(* PLC project Robots Function Blocks, JihuaLab Robots Function Blocks 1.0, author Zebang Zhong *)
(* stored: creationDateTime 2020-02-21T09:44:11, modificationDateTime 2020-04-25T15:42:12 *)

(* This block makes the robot ready. *)
FUNCTION_BLOCK RobotEnable
  VAR_INPUT
    ENABLE : BOOL;  (* TRUE to enable the block *)
    STATE : SINT;  (* Current state of robot *)
  END_VAR
  VAR_OUTPUT
    VALID : BOOL;  (* This is the output shows if robot is enabled *)
  END_VAR

          If ENABLE = TRUE then run
        
END_FUNCTION_BLOCK

(* This block makes the robot ready. *)
FUNCTION_BLOCK MotionGo
  VAR_INPUT
    ENABLE : BOOL;  (* TRUE to enable the block *)
  END_VAR
  VAR_OUTPUT
    VALID : BOOL;  (* This is the output shows if robot is ready *)
  END_VAR

          If ENABLE = TRUE then run
        
END_FUNCTION_BLOCK

(* This block gets the current joints of the robot. *)
FUNCTION_BLOCK GetCurJoint
  VAR_INPUT
    ENABLE : BOOL;  (* TRUE to enable the block *)
  END_VAR
  VAR_OUTPUT
    VALID : BOOL;  (* This is the output shows if result received *)
    ERROR : BOOL;  (* This is the output shows if error occured *)
    ERRORCODE : SINT;  (* This is the output shows the error code *)
    JOINT : STRING;  (* This is the output shows the joints *)
    EXTJOINT : STRING;  (* This is the output shows the extjoints *)
  END_VAR

          If ENABLE = TRUE then run
        
END_FUNCTION_BLOCK

(* This block gets the current state of the robot. *)
FUNCTION_BLOCK GetCurState
  VAR_INPUT
    ENABLE : BOOL;  (* TRUE to enable the block *)
  END_VAR
  VAR_OUTPUT
    STATE : SINT;  (* This is the output shows the state *)
  END_VAR

          If ENABLE = TRUE then run
        
END_FUNCTION_BLOCK

(* This block starts error recovering. *)
FUNCTION_BLOCK ErrorRecover
  VAR_INPUT
    ENABLE : BOOL;  (* TRUE to start recover *)
  END_VAR

          If ENABLE = TRUE then run
        
END_FUNCTION_BLOCK

(* This block makes the robot move. *)
FUNCTION_BLOCK MoveAbsJoint
  VAR_INPUT
    ENABLE : BOOL;  (* TRUE to enable the block *)
    JOINT : STRING;  (* This is the input of joints *)
    EXTJOINT : STRING;  (* This is the input of extjoints *)
    LOAD : STRING;  (* This is the input of load *)
    SPEED : REAL;  (* Speed of the movement *)
    ZONE : REAL;  (* Size of zone *)
  END_VAR
  VAR_OUTPUT
    VALID : BOOL;  (* This is the output shows if result received *)
    ERROR : BOOL;  (* This is the output shows if error occured *)
    ERRORCODE : SINT;  (* This is the output shows the error code *)
  END_VAR

          If ENABLE = TRUE then run
        
END_FUNCTION_BLOCK

(* This block makes the robot move. *)
FUNCTION_BLOCK MoveJoint
  VAR_INPUT
    ENABLE : BOOL;  (* TRUE to enable the block *)
    TOPOINT : STRING;  (* This is the input of target point *)
    EXTJOINT : STRING;  (* This is the input of extjoints *)
    LOAD : STRING;  (* This is the input of load *)
    SPEED : REAL;  (* Speed of the movement *)
    ZONE : REAL;  (* Size of zone *)
  END_VAR
  VAR_OUTPUT
    VALID : BOOL;  (* This is the output shows if result received *)
    ERROR : BOOL;  (* This is the output shows if error occured *)
    ERRORCODE : SINT;  (* This is the output shows the error code *)
  END_VAR

          If ENABLE = TRUE then run
        
END_FUNCTION_BLOCK

(* This block makes the robot move. *)
FUNCTION_BLOCK MoveLinear
  VAR_INPUT
    ENABLE : BOOL;  (* TRUE to enable the block *)
    TOPOINT : STRING;  (* This is the input of target point *)
    EXTJOINT : STRING;  (* This is the input of extjoints *)
    LOAD : STRING;  (* This is the input of load *)
    SPEED : REAL;  (* Speed of the movement *)
    ZONE : REAL;  (* Size of zone *)
  END_VAR
  VAR_OUTPUT
    VALID : BOOL;  (* This is the output shows if result received *)
    ERROR : BOOL;  (* This is the output shows if error occured *)
    ERRORCODE : SINT;  (* This is the output shows the error code *)
  END_VAR

          If ENABLE = TRUE then run
        
END_FUNCTION_BLOCK

(* This block makes the robot move. *)
FUNCTION_BLOCK MoveCircle
  VAR_INPUT
    ENABLE : BOOL;  (* TRUE to enable the block *)
    TOPOINT : STRING;  (* This is the input of target point *)
    EXTJOINT : STRING;  (* This is the input of extjoints *)
    VIAPOINT : STRING;  (* This is the input of via point *)
    VIAEXTJOINT : STRING;  (* This is the input of viaextjoints *)
    LOAD : STRING;  (* This is the input of load *)
    SPEED : REAL;  (* Speed of the movement *)
    ZONE : REAL;  (* Size of zone *)
  END_VAR
  VAR_OUTPUT
    VALID : BOOL;  (* This is the output shows if result received *)
    ERROR : BOOL;  (* This is the output shows if error occured *)
    ERRORCODE : SINT;  (* This is the output shows the error code *)
  END_VAR

          If ENABLE = TRUE then run
        
END_FUNCTION_BLOCK

(* This block makes the robot move. *)
FUNCTION_BLOCK MoveJogJoint
  VAR_INPUT
    ENABLE : BOOL;  (* TRUE to enable the block *)
    INDEX : SINT;  (* This is the input of the joint index *)
    LOAD : STRING;  (* This is the input of load *)
    SPEED : REAL;  (* Speed of the movement *)
  END_VAR

          If ENABLE = TRUE then run
        
END_FUNCTION_BLOCK

(* This block makes the robot move. *)
FUNCTION_BLOCK MoveJogLinear
  VAR_INPUT
    ENABLE : BOOL;  (* TRUE to enable the block *)
    JOGTYPE : SINT;  (* This is the input of the jog type *)
    LOAD : STRING;  (* This is the input of load *)
    SPEED : REAL;  (* Speed of the movement *)
  END_VAR

          If ENABLE = TRUE then run
        
END_FUNCTION_BLOCK

(* This block makes the robot move. *)
FUNCTION_BLOCK MoveJogRotation
  VAR_INPUT
    ENABLE : BOOL;  (* TRUE to enable the block *)
    JOGTYPE : SINT;  (* This is the input of the jog type *)
    LOAD : STRING;  (* This is the input of load *)
    SPEED : REAL;  (* Speed of the movement *)
  END_VAR

          If ENABLE = TRUE then run
        
END_FUNCTION_BLOCK

(* This block selects an index. *)
FUNCTION_BLOCK JogJointSelection
  VAR_INPUT
    JOINT1_F : BOOL;  (* This is the input of Joint 1 moving forward *)
    JOINT1_R : BOOL;  (* This is the input of Joint 1 moving reversed *)
    JOINT2_F : BOOL;  (* This is the input of Joint 2 moving forward *)
    JOINT2_R : BOOL;  (* This is the input of Joint 2 moving reversed *)
    JOINT3_F : BOOL;  (* This is the input of Joint 3 moving forward *)
    JOINT3_R : BOOL;  (* This is the input of Joint 3 moving reversed *)
    JOINT4_F : BOOL;  (* This is the input of Joint 4 moving forward *)
    JOINT4_R : BOOL;  (* This is the input of Joint 4 moving reversed *)
    JOINT5_F : BOOL;  (* This is the input of Joint 5 moving forward *)
    JOINT5_R : BOOL;  (* This is the input of Joint 5 moving reversed *)
    JOINT6_F : BOOL;  (* This is the input of Joint 6 moving forward *)
    JOINT6_R : BOOL;  (* This is the input of Joint 6 moving reversed *)
    IN_SPEED : REAL;  (* Speed of the movement *)
  END_VAR
  VAR_OUTPUT
    VALID : BOOL;  (* this is the output shows if input is legal *)
    INDEX : SINT;  (* this is the output of the joint index *)
    OUT_SPEED : REAL;  (* Speed of the movement *)
  END_VAR

          
        
END_FUNCTION_BLOCK

(* This block selects a jogtype. *)
FUNCTION_BLOCK JogLRSelection
  VAR_INPUT
    X_F : BOOL;  (* This is the input of moving forward along X-axis *)
    X_R : BOOL;  (* This is the input of moving backward along X-axis *)
    Y_F : BOOL;  (* This is the input of moving forward along Y-axis *)
    Y_R : BOOL;  (* This is the input of moving backword along Y-axis *)
    Z_F : BOOL;  (* This is the input of moving forward along Z-axis *)
    Z_R : BOOL;  (* This is the input of moving backword along Z-axis *)
    RX_F : BOOL;  (* This is the input of rotating forward around X-axis *)
    RX_R : BOOL;  (* This is the input of rotating backward around X-axis *)
    RY_F : BOOL;  (* This is the input of rotating forward around Y-axis *)
    RY_R : BOOL;  (* This is the input of rotating backward around Y-axis *)
    RZ_F : BOOL;  (* This is the input of rotating forward around Z-axis *)
    RZ_R : BOOL;  (* This is the input of rotating backward around X-axis *)
    IN_SPEED : REAL;  (* Speed of the movement *)
  END_VAR
  VAR_OUTPUT
    L_VALID : BOOL;  (* this is the output shows if input of MoveJogLinear is legal *)
    L_JOGTYPE : SINT;  (* This is the output of MoveJogLinear jogtype *)
    R_VALID : BOOL;  (* this is the output shows if input of MoveJogRotation is legal *)
    R_JOGTYPE : SINT;  (* This is the output of MoveJogRotation jogtype *)
    OUT_SPEED : REAL;  (* Speed of the movement *)
  END_VAR

          
        
END_FUNCTION_BLOCK

(* This block adjusts the speed of movement. *)
FUNCTION_BLOCK SpeedAdjust
  VAR_INPUT
    ACC : BOOL;  (* This is the input of accelerating speed *)
    DEC : BOOL;  (* This is the input of decelerating speed *)
  END_VAR
  VAR_OUTPUT
    SPEED : REAL;  (* Speed of the movement *)
  END_VAR

          
        
END_FUNCTION_BLOCK
